// TIA Portal V20 export
DATA_BLOCK "instFB_AxisCtrl"   // DB2
VERSION : 1.1
// stored: InstanceOfName FB_AxisCtrl, InstanceOfType FB
"FB_AxisCtrl"
   // VAR
   //    instGroupPower { S7_SetPoint := 'True'} : "LKinCtrl_MC_GroupPower";
   //    instGroupReset { S7_SetPoint := 'True'} : "LKinCtrl_MC_GroupReset";
   //    instMC_SetTool { S7_SetPoint := 'True'} : MC_SETTOOL;
   //    instMoveLinAbs : MC_MOVELINEARABSOLUTE;
   //    instJogFrame { S7_SetPoint := 'True'} : "LKinCtrl_MC_JogFrame";
   //    statToolActivated : Bool;
   // END_VAR
BEGIN
END_DATA_BLOCK
